FUNCTION_BLOCK DataPanel_xDB_16_PWM_SAE_J1939 (* Service Interface Function Block Type *)
  (* Standard: SAE J1939; Function: All Outputs: Unpaired PWM/PWM(i); Type: DP-34044-3-000 *)
  (* Version 1.0, 2018-12-05, Jose Cabral *)
  (* Version 1.0, 2022-08-04, Franz Höpfinger, Unknown *)
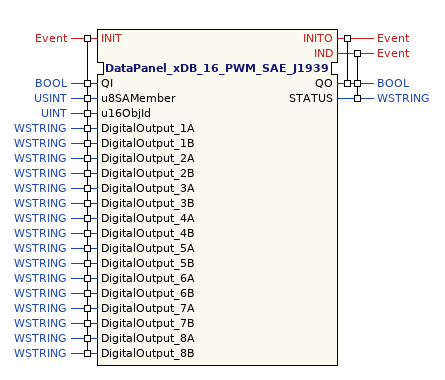
  EVENT_INPUT
    INIT WITH QI, u8SAMember, u16ObjId, DigitalOutput_1A, DigitalOutput_1B, DigitalOutput_2A, DigitalOutput_2B, DigitalOutput_3A, DigitalOutput_3B, DigitalOutput_4A, DigitalOutput_4B, DigitalOutput_5A, DigitalOutput_5B, DigitalOutput_6A, DigitalOutput_6B, DigitalOutput_7A, DigitalOutput_7B, DigitalOutput_8A, DigitalOutput_8B; (* Service Initialization *)
  END_EVENT
  EVENT_OUTPUT
    INITO WITH QO; (* Initialization Confirm *)
    IND WITH QO, STATUS; (* Indication from Resource *)
  END_EVENT
  VAR_INPUT
    QI : BOOL; (* Event Input Qualifier *)
    u8SAMember : USINT := 224; (* Node SA 224..239 *)
    u16ObjId : UINT := 65535; (* Dummy ! set to 65535 if in Doubt. 0 deactivates FB. *)
    DigitalOutput_1A : WSTRING := "DigitalOutput_1A";
    DigitalOutput_1B : WSTRING := "DigitalOutput_1B";
    DigitalOutput_2A : WSTRING := "DigitalOutput_2A";
    DigitalOutput_2B : WSTRING := "DigitalOutput_2B";
    DigitalOutput_3A : WSTRING := "DigitalOutput_3A";
    DigitalOutput_3B : WSTRING := "DigitalOutput_3B";
    DigitalOutput_4A : WSTRING := "DigitalOutput_4A";
    DigitalOutput_4B : WSTRING := "DigitalOutput_4B";
    DigitalOutput_5A : WSTRING := "DigitalOutput_5A";
    DigitalOutput_5B : WSTRING := "DigitalOutput_5B";
    DigitalOutput_6A : WSTRING := "DigitalOutput_6A";
    DigitalOutput_6B : WSTRING := "DigitalOutput_6B";
    DigitalOutput_7A : WSTRING := "DigitalOutput_7A";
    DigitalOutput_7B : WSTRING := "DigitalOutput_7B";
    DigitalOutput_8A : WSTRING := "DigitalOutput_8A";
    DigitalOutput_8B : WSTRING := "DigitalOutput_8B";
  END_VAR
  VAR_OUTPUT
    QO : BOOL; (* Event Output Qualifier *)
    STATUS : WSTRING; (* Service Status *)
  END_VAR
END_FUNCTION_BLOCK
